Universal Robots PolyScope program: pick_place.urp

Program pick_pose (installation=default directory=/home/ur/ursim-current/programs createdIn=5.14.0 lastSavedIn=5.14.0 robotSerialNumber=20195299999)
Calibrated DH parameters: a=[0, -0.6127, -0.57155, 0, 0, 0]; d=[0.1807, 0, 0, 0.17415, 0.11985, 0.11655]; alpha=[1.570796, 0, 0, 1.570796, -1.570796, 0]; deltaTheta=[0, 0, 0, 0, 0, 0]
InitVariablesNode
Robot Program (runOnlyOnce=false)
  Script file /home/ur/ursim-current/programs/pick_place.script
    | # variables
    | repetitions = 20
    | counter = 0
    | loop_forever = False
    | velocity = 200
    | status = "READY"
    | 
    | # gripper functions
    | def open_gripper():
    |     textmsg("open")
    |     #rq_open()
    | end
    | 
    | def close_gripper():
    |     textmsg("close")
    |     #rq_close()
    | end
    | 
    | # pick place functions
    | def pick(pose):
    |     status = "PICKING"
    |     approach = pose_trans(pose, p[0, 0, -0.1, 0, 0, 0])
    |     movel(approach, a=0.1, v=velocity/1000)
    |     movel(pick_pose, a=0.1, v=velocity/1000)
    |     close_gripper()
    |     movel(approach, a=0.1, v=velocity/1000)
    | end
    | 
    | def place(pose):
    |     status = "PLACING"
    |     approach = pose_trans(pose, p[0, 0, -0.1, 0, 0, 0])
    |     movel(approach, a=0.1, v=velocity/1000)
    |     movel(pick_pose, a=0.1, v=velocity/1000)
    |     open_gripper()
    |     movel(approach, a=0.1, v=velocity/1000)
    | end
    | 
    | def start_task():
    |     while loop_forever or counter < repetitions:
    |         pick(pick_pose)
    |         place(place_pose)
    |         pick(place_pose)
    |         place(pick_pose)
    |         counter = counter + 1
    |     end
    |     status = "READY"
    | end
  URCap HMI (Robpod HMI URcap, Robpod Cloud) dataModel(robpod.hmi.selected=/home/ur/ursim-current/programs/pick_place.hmi, robpod.hmi.stop.main.loop=true)
